// TIA Portal V20 export
FUNCTION_BLOCK "Count"   // FB22, LAD
// stored: MemoryReserve 100, SetENOAutomatically false
   VAR
      statPulse { ExternalAccessible := 'False'; ExternalVisible := 'False'; ExternalWritable := 'False'} : Array[0..299] of Bool;
   END_VAR
   VAR_TEMP   // added for the SCL form of the ladder/FBD networks
      _w1 : Bool;
      _w2 : Bool;
      _w3 : Bool;
   END_VAR
BEGIN

REGION Network 1 (SCL): Alarms Count l Button
   // Alarm Save
   IF "Unit1.Em3.HmiInterface".topTapeCuttingCount.alarmSaveButton THEN
       "Unit1.Em3.HmiInterface".topTapeCuttingCount.ProcessValue.warningCount := "Unit1.Em3.HmiInterface".topTapeCuttingCount.SetValue.warningCount;
       "Unit1.Em3.HmiInterface".topTapeCuttingCount.ProcessValue.faultCount := "Unit1.Em3.HmiInterface".topTapeCuttingCount.SetValue.faultCount;
   END_IF;
   IF "Unit1.Em4.HmiInterface".sideTapeCuttingCount.alarmSaveButton THEN
       "Unit1.Em4.HmiInterface".sideTapeCuttingCount.ProcessValue.warningCount := "Unit1.Em4.HmiInterface".sideTapeCuttingCount.SetValue.warningCount;
       "Unit1.Em4.HmiInterface".sideTapeCuttingCount.ProcessValue.faultCount := "Unit1.Em4.HmiInterface".sideTapeCuttingCount.SetValue.faultCount;
   END_IF;
   IF "Unit1.Em9.HmiInterface".VisionNgAlarmCount.alarmSaveButton THEN
       "Unit1.Em9.HmiInterface".VisionNgAlarmCount.ProcessValue.warningCount:= "Unit1.Em9.HmiInterface".VisionNgAlarmCount.SetValue.warningCount;
       "Unit1.Em9.HmiInterface".VisionNgAlarmCount.ProcessValue.faultCount := "Unit1.Em9.HmiInterface".VisionNgAlarmCount.SetValue.faultCount;
   END_IF;


   // Count Reset
   IF "Unit1.Em3.HmiInterface".topTapeCuttingCount.countResetButton THEN
       "Unit1.Em3.HmiInterface".topTapeCuttingCount.actualCount := 0;
   END_IF;
   IF "Unit1.Em4.HmiInterface".sideTapeCuttingCount.countResetButton THEN
       "Unit1.Em4.HmiInterface".sideTapeCuttingCount.actualCount := 0;
   END_IF;
   IF "Unit1.Em9.HmiInterface".VisionNgAlarmCount.countResetButton THEN
       "Unit1.Em9.HmiInterface".VisionNgAlarmCount.actualCount := 0;
   END_IF;
END_REGION

REGION Network 2: Alarms Count l Top Tape Cutting Count Up
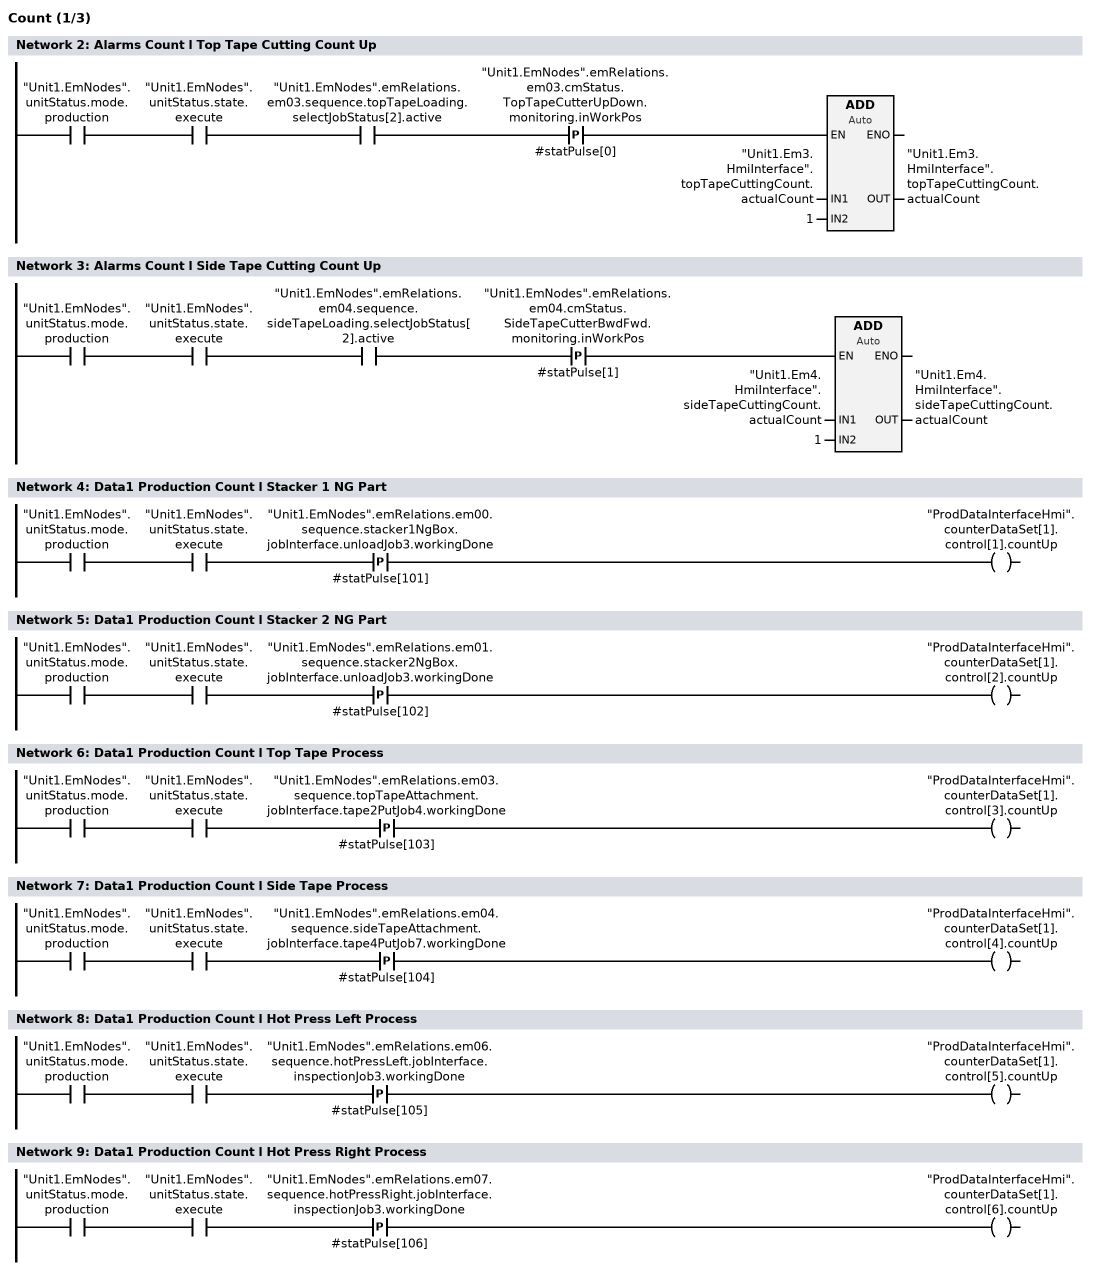
   RUNG wire#powerrail
      Contact( "Unit1.EmNodes".unitStatus.mode.production )
      Contact( "Unit1.EmNodes".unitStatus.state.execute )
      Contact( "Unit1.EmNodes".emRelations.em03.sequence.topTapeLoading.selectJobStatus[2].active )
      P_Contact(operand := "Unit1.EmNodes".emRelations.em03.cmStatus.TopTapeCutterUpDown.monitoring.inWorkPos, bit := #statPulse[0])
      Add(in1 := "Unit1.Em3.HmiInterface".topTapeCuttingCount.actualCount, in2 := 1, out => "Unit1.Em3.HmiInterface".topTapeCuttingCount.actualCount)
   END_RUNG
   // the same network as SCL:
   #_w1 := "Unit1.EmNodes".unitStatus.mode.production AND "Unit1.EmNodes".unitStatus.state.execute AND "Unit1.EmNodes".emRelations.em03.sequence.topTapeLoading.selectJobStatus[2].active AND "Unit1.EmNodes".emRelations.em03.cmStatus.TopTapeCutterUpDown.monitoring.inWorkPos AND NOT #statPulse[0];   // rising edge of "Unit1.EmNodes".emRelations.em03.cmStatus.TopTapeCutterUpDown.monitoring.inWorkPos
   #statPulse[0] := "Unit1.EmNodes".emRelations.em03.cmStatus.TopTapeCutterUpDown.monitoring.inWorkPos;
   IF #_w1 THEN
       "Unit1.Em3.HmiInterface".topTapeCuttingCount.actualCount := "Unit1.Em3.HmiInterface".topTapeCuttingCount.actualCount + 1;
   END_IF;
END_REGION

REGION Network 3: Alarms Count l Side Tape Cutting Count Up
   RUNG wire#powerrail
      Contact( "Unit1.EmNodes".unitStatus.mode.production )
      Contact( "Unit1.EmNodes".unitStatus.state.execute )
      Contact( "Unit1.EmNodes".emRelations.em04.sequence.sideTapeLoading.selectJobStatus[2].active )
      P_Contact(operand := "Unit1.EmNodes".emRelations.em04.cmStatus.SideTapeCutterBwdFwd.monitoring.inWorkPos, bit := #statPulse[1])
      Add(in1 := "Unit1.Em4.HmiInterface".sideTapeCuttingCount.actualCount, in2 := 1, out => "Unit1.Em4.HmiInterface".sideTapeCuttingCount.actualCount)
   END_RUNG
   // the same network as SCL:
   #_w1 := "Unit1.EmNodes".unitStatus.mode.production AND "Unit1.EmNodes".unitStatus.state.execute AND "Unit1.EmNodes".emRelations.em04.sequence.sideTapeLoading.selectJobStatus[2].active AND "Unit1.EmNodes".emRelations.em04.cmStatus.SideTapeCutterBwdFwd.monitoring.inWorkPos AND NOT #statPulse[1];   // rising edge of "Unit1.EmNodes".emRelations.em04.cmStatus.SideTapeCutterBwdFwd.monitoring.inWorkPos
   #statPulse[1] := "Unit1.EmNodes".emRelations.em04.cmStatus.SideTapeCutterBwdFwd.monitoring.inWorkPos;
   IF #_w1 THEN
       "Unit1.Em4.HmiInterface".sideTapeCuttingCount.actualCount := "Unit1.Em4.HmiInterface".sideTapeCuttingCount.actualCount + 1;
   END_IF;
END_REGION

REGION Network 4: Data1 Production Count l Stacker 1 NG Part
   RUNG wire#powerrail
      Contact( "Unit1.EmNodes".unitStatus.mode.production )
      Contact( "Unit1.EmNodes".unitStatus.state.execute )
      P_Contact(operand := "Unit1.EmNodes".emRelations.em00.sequence.stacker1NgBox.jobInterface.unloadJob3.workingDone, bit := #statPulse[101])
      Coil( "ProdDataInterfaceHmi".counterDataSet[1].control[1].countUp )
   END_RUNG
   // the same network as SCL:
   #_w1 := "Unit1.EmNodes".unitStatus.mode.production AND "Unit1.EmNodes".unitStatus.state.execute AND "Unit1.EmNodes".emRelations.em00.sequence.stacker1NgBox.jobInterface.unloadJob3.workingDone AND NOT #statPulse[101];   // rising edge of "Unit1.EmNodes".emRelations.em00.sequence.stacker1NgBox.jobInterface.unloadJob3.workingDone
   #statPulse[101] := "Unit1.EmNodes".emRelations.em00.sequence.stacker1NgBox.jobInterface.unloadJob3.workingDone;
   "ProdDataInterfaceHmi".counterDataSet[1].control[1].countUp := #_w1;
END_REGION

REGION Network 5: Data1 Production Count l Stacker 2 NG Part
   RUNG wire#powerrail
      Contact( "Unit1.EmNodes".unitStatus.mode.production )
      Contact( "Unit1.EmNodes".unitStatus.state.execute )
      P_Contact(operand := "Unit1.EmNodes".emRelations.em01.sequence.stacker2NgBox.jobInterface.unloadJob3.workingDone, bit := #statPulse[102])
      Coil( "ProdDataInterfaceHmi".counterDataSet[1].control[2].countUp )
   END_RUNG
   // the same network as SCL:
   #_w1 := "Unit1.EmNodes".unitStatus.mode.production AND "Unit1.EmNodes".unitStatus.state.execute AND "Unit1.EmNodes".emRelations.em01.sequence.stacker2NgBox.jobInterface.unloadJob3.workingDone AND NOT #statPulse[102];   // rising edge of "Unit1.EmNodes".emRelations.em01.sequence.stacker2NgBox.jobInterface.unloadJob3.workingDone
   #statPulse[102] := "Unit1.EmNodes".emRelations.em01.sequence.stacker2NgBox.jobInterface.unloadJob3.workingDone;
   "ProdDataInterfaceHmi".counterDataSet[1].control[2].countUp := #_w1;
END_REGION

REGION Network 6: Data1 Production Count l Top Tape Process
   RUNG wire#powerrail
      Contact( "Unit1.EmNodes".unitStatus.mode.production )
      Contact( "Unit1.EmNodes".unitStatus.state.execute )
      P_Contact(operand := "Unit1.EmNodes".emRelations.em03.sequence.topTapeAttachment.jobInterface.tape2PutJob4.workingDone, bit := #statPulse[103])
      Coil( "ProdDataInterfaceHmi".counterDataSet[1].control[3].countUp )
   END_RUNG
   // the same network as SCL:
   #_w1 := "Unit1.EmNodes".unitStatus.mode.production AND "Unit1.EmNodes".unitStatus.state.execute AND "Unit1.EmNodes".emRelations.em03.sequence.topTapeAttachment.jobInterface.tape2PutJob4.workingDone AND NOT #statPulse[103];   // rising edge of "Unit1.EmNodes".emRelations.em03.sequence.topTapeAttachment.jobInterface.tape2PutJob4.workingDone
   #statPulse[103] := "Unit1.EmNodes".emRelations.em03.sequence.topTapeAttachment.jobInterface.tape2PutJob4.workingDone;
   "ProdDataInterfaceHmi".counterDataSet[1].control[3].countUp := #_w1;
END_REGION

REGION Network 7: Data1 Production Count l Side Tape Process
   RUNG wire#powerrail
      Contact( "Unit1.EmNodes".unitStatus.mode.production )
      Contact( "Unit1.EmNodes".unitStatus.state.execute )
      P_Contact(operand := "Unit1.EmNodes".emRelations.em04.sequence.sideTapeAttachment.jobInterface.tape4PutJob7.workingDone, bit := #statPulse[104])
      Coil( "ProdDataInterfaceHmi".counterDataSet[1].control[4].countUp )
   END_RUNG
   // the same network as SCL:
   #_w1 := "Unit1.EmNodes".unitStatus.mode.production AND "Unit1.EmNodes".unitStatus.state.execute AND "Unit1.EmNodes".emRelations.em04.sequence.sideTapeAttachment.jobInterface.tape4PutJob7.workingDone AND NOT #statPulse[104];   // rising edge of "Unit1.EmNodes".emRelations.em04.sequence.sideTapeAttachment.jobInterface.tape4PutJob7.workingDone
   #statPulse[104] := "Unit1.EmNodes".emRelations.em04.sequence.sideTapeAttachment.jobInterface.tape4PutJob7.workingDone;
   "ProdDataInterfaceHmi".counterDataSet[1].control[4].countUp := #_w1;
END_REGION

REGION Network 8: Data1 Production Count l Hot Press Left Process
   RUNG wire#powerrail
      Contact( "Unit1.EmNodes".unitStatus.mode.production )
      Contact( "Unit1.EmNodes".unitStatus.state.execute )
      P_Contact(operand := "Unit1.EmNodes".emRelations.em06.sequence.hotPressLeft.jobInterface.inspectionJob3.workingDone, bit := #statPulse[105])
      Coil( "ProdDataInterfaceHmi".counterDataSet[1].control[5].countUp )
   END_RUNG
   // the same network as SCL:
   #_w1 := "Unit1.EmNodes".unitStatus.mode.production AND "Unit1.EmNodes".unitStatus.state.execute AND "Unit1.EmNodes".emRelations.em06.sequence.hotPressLeft.jobInterface.inspectionJob3.workingDone AND NOT #statPulse[105];   // rising edge of "Unit1.EmNodes".emRelations.em06.sequence.hotPressLeft.jobInterface.inspectionJob3.workingDone
   #statPulse[105] := "Unit1.EmNodes".emRelations.em06.sequence.hotPressLeft.jobInterface.inspectionJob3.workingDone;
   "ProdDataInterfaceHmi".counterDataSet[1].control[5].countUp := #_w1;
END_REGION

REGION Network 9: Data1 Production Count l Hot Press Right Process
   RUNG wire#powerrail
      Contact( "Unit1.EmNodes".unitStatus.mode.production )
      Contact( "Unit1.EmNodes".unitStatus.state.execute )
      P_Contact(operand := "Unit1.EmNodes".emRelations.em07.sequence.hotPressRight.jobInterface.inspectionJob3.workingDone, bit := #statPulse[106])
      Coil( "ProdDataInterfaceHmi".counterDataSet[1].control[6].countUp )
   END_RUNG
   // the same network as SCL:
   #_w1 := "Unit1.EmNodes".unitStatus.mode.production AND "Unit1.EmNodes".unitStatus.state.execute AND "Unit1.EmNodes".emRelations.em07.sequence.hotPressRight.jobInterface.inspectionJob3.workingDone AND NOT #statPulse[106];   // rising edge of "Unit1.EmNodes".emRelations.em07.sequence.hotPressRight.jobInterface.inspectionJob3.workingDone
   #statPulse[106] := "Unit1.EmNodes".emRelations.em07.sequence.hotPressRight.jobInterface.inspectionJob3.workingDone;
   "ProdDataInterfaceHmi".counterDataSet[1].control[6].countUp := #_w1;
END_REGION

REGION Network 10: Data1 Production Count l Hipot & Thickness Servo Press Process
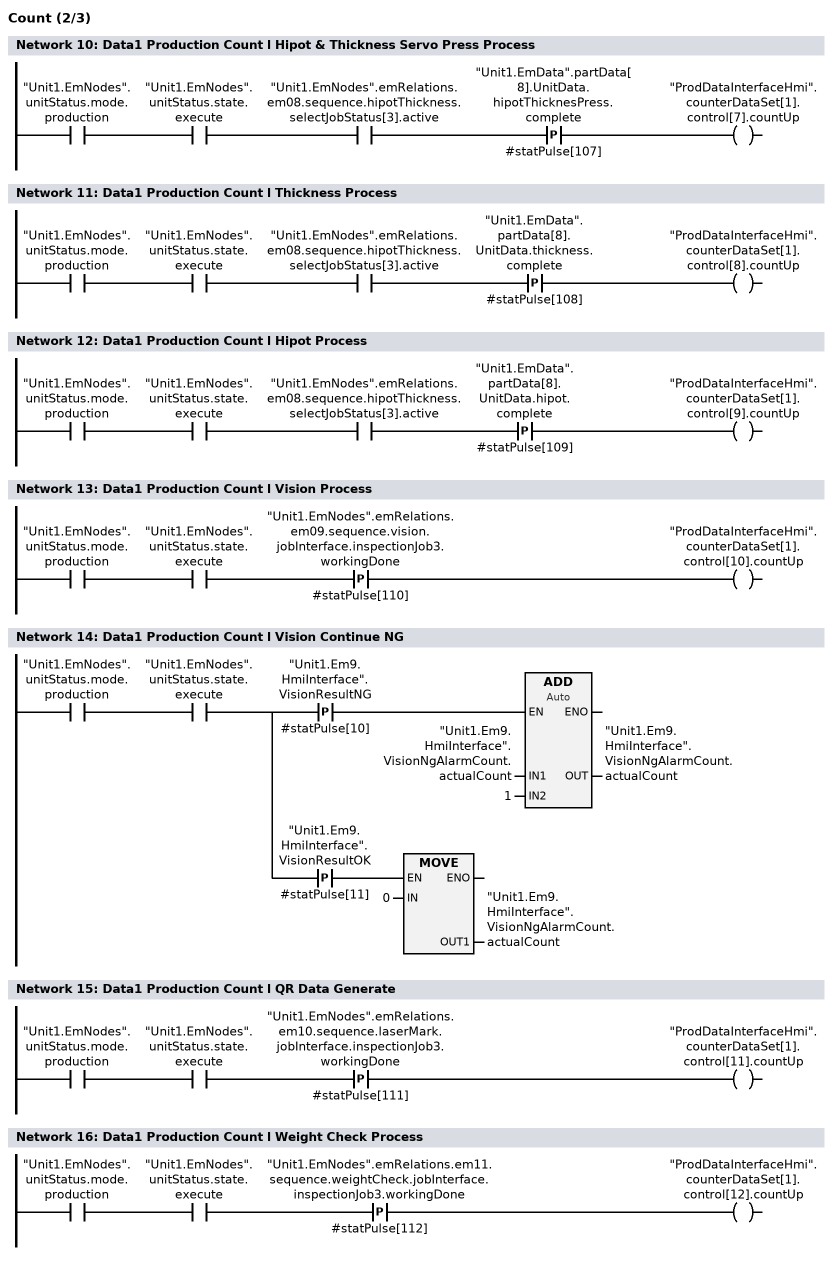
   RUNG wire#powerrail
      Contact( "Unit1.EmNodes".unitStatus.mode.production )
      Contact( "Unit1.EmNodes".unitStatus.state.execute )
      Contact( "Unit1.EmNodes".emRelations.em08.sequence.hipotThickness.selectJobStatus[3].active )
      P_Contact(operand := "Unit1.EmData".partData[8].UnitData.hipotThicknesPress.complete, bit := #statPulse[107])
      Coil( "ProdDataInterfaceHmi".counterDataSet[1].control[7].countUp )
   END_RUNG
   // the same network as SCL:
   #_w1 := "Unit1.EmNodes".unitStatus.mode.production AND "Unit1.EmNodes".unitStatus.state.execute AND "Unit1.EmNodes".emRelations.em08.sequence.hipotThickness.selectJobStatus[3].active AND "Unit1.EmData".partData[8].UnitData.hipotThicknesPress.complete AND NOT #statPulse[107];   // rising edge of "Unit1.EmData".partData[8].UnitData.hipotThicknesPress.complete
   #statPulse[107] := "Unit1.EmData".partData[8].UnitData.hipotThicknesPress.complete;
   "ProdDataInterfaceHmi".counterDataSet[1].control[7].countUp := #_w1;
END_REGION

REGION Network 11: Data1 Production Count l Thickness Process
   RUNG wire#powerrail
      Contact( "Unit1.EmNodes".unitStatus.mode.production )
      Contact( "Unit1.EmNodes".unitStatus.state.execute )
      Contact( "Unit1.EmNodes".emRelations.em08.sequence.hipotThickness.selectJobStatus[3].active )
      P_Contact(operand := "Unit1.EmData".partData[8].UnitData.thickness.complete, bit := #statPulse[108])
      Coil( "ProdDataInterfaceHmi".counterDataSet[1].control[8].countUp )
   END_RUNG
   // the same network as SCL:
   #_w1 := "Unit1.EmNodes".unitStatus.mode.production AND "Unit1.EmNodes".unitStatus.state.execute AND "Unit1.EmNodes".emRelations.em08.sequence.hipotThickness.selectJobStatus[3].active AND "Unit1.EmData".partData[8].UnitData.thickness.complete AND NOT #statPulse[108];   // rising edge of "Unit1.EmData".partData[8].UnitData.thickness.complete
   #statPulse[108] := "Unit1.EmData".partData[8].UnitData.thickness.complete;
   "ProdDataInterfaceHmi".counterDataSet[1].control[8].countUp := #_w1;
END_REGION

REGION Network 12: Data1 Production Count l Hipot Process
   RUNG wire#powerrail
      Contact( "Unit1.EmNodes".unitStatus.mode.production )
      Contact( "Unit1.EmNodes".unitStatus.state.execute )
      Contact( "Unit1.EmNodes".emRelations.em08.sequence.hipotThickness.selectJobStatus[3].active )
      P_Contact(operand := "Unit1.EmData".partData[8].UnitData.hipot.complete, bit := #statPulse[109])
      Coil( "ProdDataInterfaceHmi".counterDataSet[1].control[9].countUp )
   END_RUNG
   // the same network as SCL:
   #_w1 := "Unit1.EmNodes".unitStatus.mode.production AND "Unit1.EmNodes".unitStatus.state.execute AND "Unit1.EmNodes".emRelations.em08.sequence.hipotThickness.selectJobStatus[3].active AND "Unit1.EmData".partData[8].UnitData.hipot.complete AND NOT #statPulse[109];   // rising edge of "Unit1.EmData".partData[8].UnitData.hipot.complete
   #statPulse[109] := "Unit1.EmData".partData[8].UnitData.hipot.complete;
   "ProdDataInterfaceHmi".counterDataSet[1].control[9].countUp := #_w1;
END_REGION

REGION Network 13: Data1 Production Count l Vision Process
   RUNG wire#powerrail
      Contact( "Unit1.EmNodes".unitStatus.mode.production )
      Contact( "Unit1.EmNodes".unitStatus.state.execute )
      P_Contact(operand := "Unit1.EmNodes".emRelations.em09.sequence.vision.jobInterface.inspectionJob3.workingDone, bit := #statPulse[110])
      Coil( "ProdDataInterfaceHmi".counterDataSet[1].control[10].countUp )
   END_RUNG
   // the same network as SCL:
   #_w1 := "Unit1.EmNodes".unitStatus.mode.production AND "Unit1.EmNodes".unitStatus.state.execute AND "Unit1.EmNodes".emRelations.em09.sequence.vision.jobInterface.inspectionJob3.workingDone AND NOT #statPulse[110];   // rising edge of "Unit1.EmNodes".emRelations.em09.sequence.vision.jobInterface.inspectionJob3.workingDone
   #statPulse[110] := "Unit1.EmNodes".emRelations.em09.sequence.vision.jobInterface.inspectionJob3.workingDone;
   "ProdDataInterfaceHmi".counterDataSet[1].control[10].countUp := #_w1;
END_REGION

REGION Network 14: Data1 Production Count l Vision Continue NG
   RUNG wire#powerrail
      Contact( "Unit1.EmNodes".unitStatus.mode.production )
      Contact( "Unit1.EmNodes".unitStatus.state.execute )
      wire#w1
      P_Contact(operand := "Unit1.Em9.HmiInterface".VisionResultNG, bit := #statPulse[10])
      Add(in1 := "Unit1.Em9.HmiInterface".VisionNgAlarmCount.actualCount, in2 := 1, out => "Unit1.Em9.HmiInterface".VisionNgAlarmCount.actualCount)
   END_RUNG
   RUNG wire#w1
      P_Contact(operand := "Unit1.Em9.HmiInterface".VisionResultOK, bit := #statPulse[11])
      Move(in := 0, out1 => "Unit1.Em9.HmiInterface".VisionNgAlarmCount.actualCount)
   END_RUNG
   // the same network as SCL:
   #_w1 := "Unit1.EmNodes".unitStatus.mode.production AND "Unit1.EmNodes".unitStatus.state.execute;
   #_w2 := #_w1 AND "Unit1.Em9.HmiInterface".VisionResultNG AND NOT #statPulse[10];   // rising edge of "Unit1.Em9.HmiInterface".VisionResultNG
   #statPulse[10] := "Unit1.Em9.HmiInterface".VisionResultNG;
   IF #_w2 THEN
       "Unit1.Em9.HmiInterface".VisionNgAlarmCount.actualCount := "Unit1.Em9.HmiInterface".VisionNgAlarmCount.actualCount + 1;
   END_IF;
   #_w3 := #_w1 AND "Unit1.Em9.HmiInterface".VisionResultOK AND NOT #statPulse[11];   // rising edge of "Unit1.Em9.HmiInterface".VisionResultOK
   #statPulse[11] := "Unit1.Em9.HmiInterface".VisionResultOK;
   IF #_w3 THEN "Unit1.Em9.HmiInterface".VisionNgAlarmCount.actualCount := 0; END_IF;
END_REGION

REGION Network 15: Data1 Production Count l QR Data Generate
   RUNG wire#powerrail
      Contact( "Unit1.EmNodes".unitStatus.mode.production )
      Contact( "Unit1.EmNodes".unitStatus.state.execute )
      P_Contact(operand := "Unit1.EmNodes".emRelations.em10.sequence.laserMark.jobInterface.inspectionJob3.workingDone, bit := #statPulse[111])
      Coil( "ProdDataInterfaceHmi".counterDataSet[1].control[11].countUp )
   END_RUNG
   // the same network as SCL:
   #_w1 := "Unit1.EmNodes".unitStatus.mode.production AND "Unit1.EmNodes".unitStatus.state.execute AND "Unit1.EmNodes".emRelations.em10.sequence.laserMark.jobInterface.inspectionJob3.workingDone AND NOT #statPulse[111];   // rising edge of "Unit1.EmNodes".emRelations.em10.sequence.laserMark.jobInterface.inspectionJob3.workingDone
   #statPulse[111] := "Unit1.EmNodes".emRelations.em10.sequence.laserMark.jobInterface.inspectionJob3.workingDone;
   "ProdDataInterfaceHmi".counterDataSet[1].control[11].countUp := #_w1;
END_REGION

REGION Network 16: Data1 Production Count l Weight Check Process
   RUNG wire#powerrail
      Contact( "Unit1.EmNodes".unitStatus.mode.production )
      Contact( "Unit1.EmNodes".unitStatus.state.execute )
      P_Contact(operand := "Unit1.EmNodes".emRelations.em11.sequence.weightCheck.jobInterface.inspectionJob3.workingDone, bit := #statPulse[112])
      Coil( "ProdDataInterfaceHmi".counterDataSet[1].control[12].countUp )
   END_RUNG
   // the same network as SCL:
   #_w1 := "Unit1.EmNodes".unitStatus.mode.production AND "Unit1.EmNodes".unitStatus.state.execute AND "Unit1.EmNodes".emRelations.em11.sequence.weightCheck.jobInterface.inspectionJob3.workingDone AND NOT #statPulse[112];   // rising edge of "Unit1.EmNodes".emRelations.em11.sequence.weightCheck.jobInterface.inspectionJob3.workingDone
   #statPulse[112] := "Unit1.EmNodes".emRelations.em11.sequence.weightCheck.jobInterface.inspectionJob3.workingDone;
   "ProdDataInterfaceHmi".counterDataSet[1].control[12].countUp := #_w1;
END_REGION

REGION Network 17: Data1 Production Count l Final NG Part
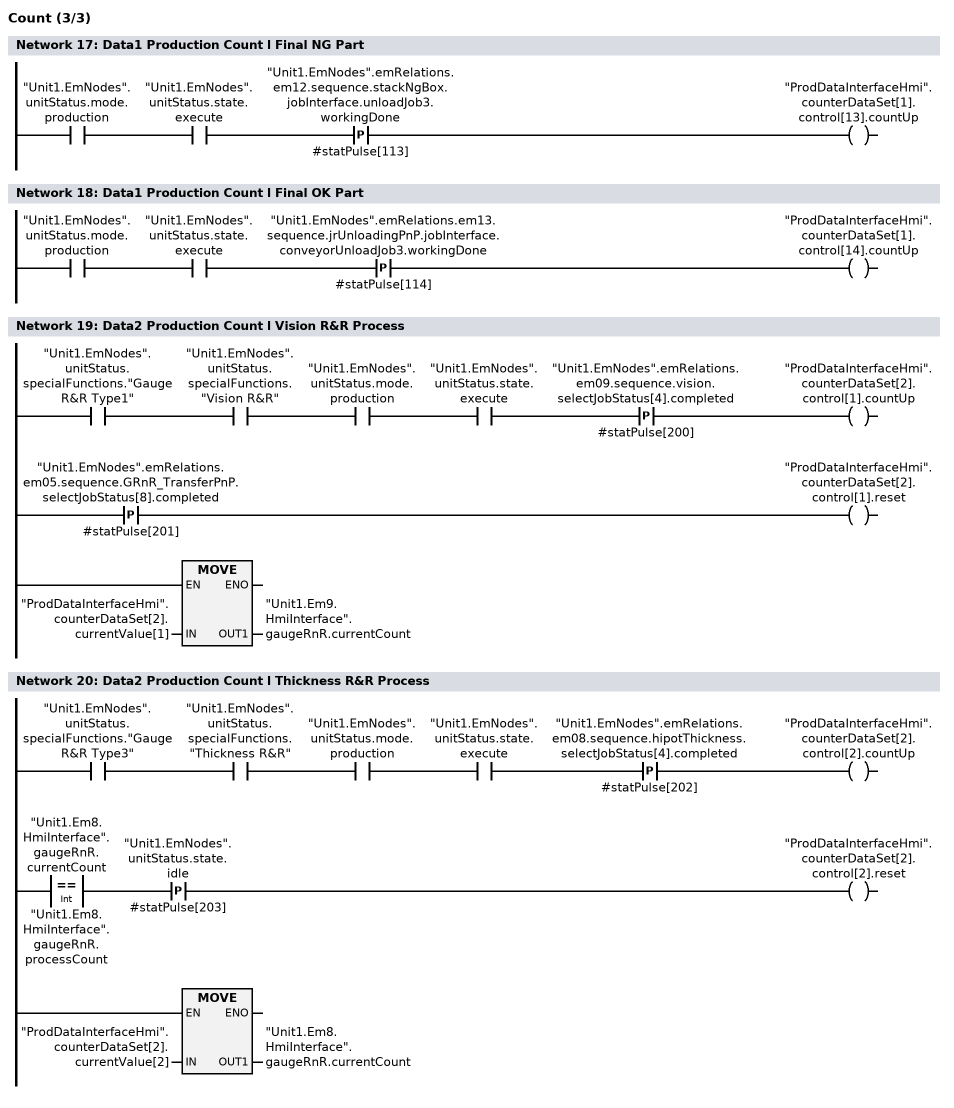
   RUNG wire#powerrail
      Contact( "Unit1.EmNodes".unitStatus.mode.production )
      Contact( "Unit1.EmNodes".unitStatus.state.execute )
      P_Contact(operand := "Unit1.EmNodes".emRelations.em12.sequence.stackNgBox.jobInterface.unloadJob3.workingDone, bit := #statPulse[113])
      Coil( "ProdDataInterfaceHmi".counterDataSet[1].control[13].countUp )
   END_RUNG
   // the same network as SCL:
   #_w1 := "Unit1.EmNodes".unitStatus.mode.production AND "Unit1.EmNodes".unitStatus.state.execute AND "Unit1.EmNodes".emRelations.em12.sequence.stackNgBox.jobInterface.unloadJob3.workingDone AND NOT #statPulse[113];   // rising edge of "Unit1.EmNodes".emRelations.em12.sequence.stackNgBox.jobInterface.unloadJob3.workingDone
   #statPulse[113] := "Unit1.EmNodes".emRelations.em12.sequence.stackNgBox.jobInterface.unloadJob3.workingDone;
   "ProdDataInterfaceHmi".counterDataSet[1].control[13].countUp := #_w1;
END_REGION

REGION Network 18: Data1 Production Count l Final OK Part
   RUNG wire#powerrail
      Contact( "Unit1.EmNodes".unitStatus.mode.production )
      Contact( "Unit1.EmNodes".unitStatus.state.execute )
      P_Contact(operand := "Unit1.EmNodes".emRelations.em13.sequence.jrUnloadingPnP.jobInterface.conveyorUnloadJob3.workingDone, bit := #statPulse[114])
      Coil( "ProdDataInterfaceHmi".counterDataSet[1].control[14].countUp )
   END_RUNG
   // the same network as SCL:
   #_w1 := "Unit1.EmNodes".unitStatus.mode.production AND "Unit1.EmNodes".unitStatus.state.execute AND "Unit1.EmNodes".emRelations.em13.sequence.jrUnloadingPnP.jobInterface.conveyorUnloadJob3.workingDone AND NOT #statPulse[114];   // rising edge of "Unit1.EmNodes".emRelations.em13.sequence.jrUnloadingPnP.jobInterface.conveyorUnloadJob3.workingDone
   #statPulse[114] := "Unit1.EmNodes".emRelations.em13.sequence.jrUnloadingPnP.jobInterface.conveyorUnloadJob3.workingDone;
   "ProdDataInterfaceHmi".counterDataSet[1].control[14].countUp := #_w1;
END_REGION

REGION Network 19: Data2 Production Count l Vision R&R Process
   RUNG wire#powerrail
      Contact( "Unit1.EmNodes".unitStatus.specialFunctions."Gauge R&R Type1" )
      Contact( "Unit1.EmNodes".unitStatus.specialFunctions."Vision R&R" )
      Contact( "Unit1.EmNodes".unitStatus.mode.production )
      Contact( "Unit1.EmNodes".unitStatus.state.execute )
      P_Contact(operand := "Unit1.EmNodes".emRelations.em09.sequence.vision.selectJobStatus[4].completed, bit := #statPulse[200])
      Coil( "ProdDataInterfaceHmi".counterDataSet[2].control[1].countUp )
   END_RUNG
   RUNG wire#powerrail
      P_Contact(operand := "Unit1.EmNodes".emRelations.em05.sequence.GRnR_TransferPnP.selectJobStatus[8].completed, bit := #statPulse[201])
      Coil( "ProdDataInterfaceHmi".counterDataSet[2].control[1].reset )
   END_RUNG
   RUNG wire#powerrail
      Move(in := "ProdDataInterfaceHmi".counterDataSet[2].currentValue[1], out1 => "Unit1.Em9.HmiInterface".gaugeRnR.currentCount)
   END_RUNG
   // the same network as SCL:
   #_w1 := "Unit1.EmNodes".unitStatus.specialFunctions."Gauge R&R Type1" AND "Unit1.EmNodes".unitStatus.specialFunctions."Vision R&R" AND "Unit1.EmNodes".unitStatus.mode.production AND "Unit1.EmNodes".unitStatus.state.execute AND "Unit1.EmNodes".emRelations.em09.sequence.vision.selectJobStatus[4].completed AND NOT #statPulse[200];   // rising edge of "Unit1.EmNodes".emRelations.em09.sequence.vision.selectJobStatus[4].completed
   #statPulse[200] := "Unit1.EmNodes".emRelations.em09.sequence.vision.selectJobStatus[4].completed;
   "ProdDataInterfaceHmi".counterDataSet[2].control[1].countUp := #_w1;
   #_w2 := "Unit1.EmNodes".emRelations.em05.sequence.GRnR_TransferPnP.selectJobStatus[8].completed AND NOT #statPulse[201];   // rising edge of "Unit1.EmNodes".emRelations.em05.sequence.GRnR_TransferPnP.selectJobStatus[8].completed
   #statPulse[201] := "Unit1.EmNodes".emRelations.em05.sequence.GRnR_TransferPnP.selectJobStatus[8].completed;
   "ProdDataInterfaceHmi".counterDataSet[2].control[1].reset := #_w2;
   "Unit1.Em9.HmiInterface".gaugeRnR.currentCount := "ProdDataInterfaceHmi".counterDataSet[2].currentValue[1];
END_REGION

REGION Network 20: Data2 Production Count l Thickness R&R Process
   RUNG wire#powerrail
      Contact( "Unit1.EmNodes".unitStatus.specialFunctions."Gauge R&R Type3" )
      Contact( "Unit1.EmNodes".unitStatus.specialFunctions."Thickness R&R" )
      Contact( "Unit1.EmNodes".unitStatus.mode.production )
      Contact( "Unit1.EmNodes".unitStatus.state.execute )
      P_Contact(operand := "Unit1.EmNodes".emRelations.em08.sequence.hipotThickness.selectJobStatus[4].completed, bit := #statPulse[202])
      Coil( "ProdDataInterfaceHmi".counterDataSet[2].control[2].countUp )
   END_RUNG
   RUNG wire#powerrail
      { S7_Templates := "SrcType := Int" } EQ_Contact(in1 := "Unit1.Em8.HmiInterface".gaugeRnR.currentCount, in2 := "Unit1.Em8.HmiInterface".gaugeRnR.processCount)
      P_Contact(operand := "Unit1.EmNodes".unitStatus.state.idle, bit := #statPulse[203])
      Coil( "ProdDataInterfaceHmi".counterDataSet[2].control[2].reset )
   END_RUNG
   RUNG wire#powerrail
      Move(in := "ProdDataInterfaceHmi".counterDataSet[2].currentValue[2], out1 => "Unit1.Em8.HmiInterface".gaugeRnR.currentCount)
   END_RUNG
   // the same network as SCL:
   #_w1 := "Unit1.EmNodes".unitStatus.specialFunctions."Gauge R&R Type3" AND "Unit1.EmNodes".unitStatus.specialFunctions."Thickness R&R" AND "Unit1.EmNodes".unitStatus.mode.production AND "Unit1.EmNodes".unitStatus.state.execute AND "Unit1.EmNodes".emRelations.em08.sequence.hipotThickness.selectJobStatus[4].completed AND NOT #statPulse[202];   // rising edge of "Unit1.EmNodes".emRelations.em08.sequence.hipotThickness.selectJobStatus[4].completed
   #statPulse[202] := "Unit1.EmNodes".emRelations.em08.sequence.hipotThickness.selectJobStatus[4].completed;
   "ProdDataInterfaceHmi".counterDataSet[2].control[2].countUp := #_w1;
   #_w2 := ("Unit1.Em8.HmiInterface".gaugeRnR.currentCount = "Unit1.Em8.HmiInterface".gaugeRnR.processCount) AND "Unit1.EmNodes".unitStatus.state.idle AND NOT #statPulse[203];   // rising edge of "Unit1.EmNodes".unitStatus.state.idle
   #statPulse[203] := "Unit1.EmNodes".unitStatus.state.idle;
   "ProdDataInterfaceHmi".counterDataSet[2].control[2].reset := #_w2;
   "Unit1.Em8.HmiInterface".gaugeRnR.currentCount := "ProdDataInterfaceHmi".counterDataSet[2].currentValue[2];
END_REGION
END_FUNCTION_BLOCK
